// TIA Portal V21 export
VAR_GLOBAL   // PLC tag table "K_Valvola_GruppoRiempi"
END_VAR
VAR_GLOBAL CONSTANT   // user constants
   K_Valvola_GruppoRiempi_Canstop : Int := 0;
END_VAR
